TEXTLIST E_Locations
  0 = 'Main PLC'
  1 = '230V Main supply'
  2 = '24V Main supply'
  3 = 'Main air supply'
  4 = 'Main Screen'
  5 = 'Main IO'
   = ''
END_TEXTLIST

(* stored: Version 1.1.0.1, ProductVersion 3.1.4024.3
   TextList E_Locations: Id {0dc60658-fd27-49a2-a55d-b05b07e19b19} *)
